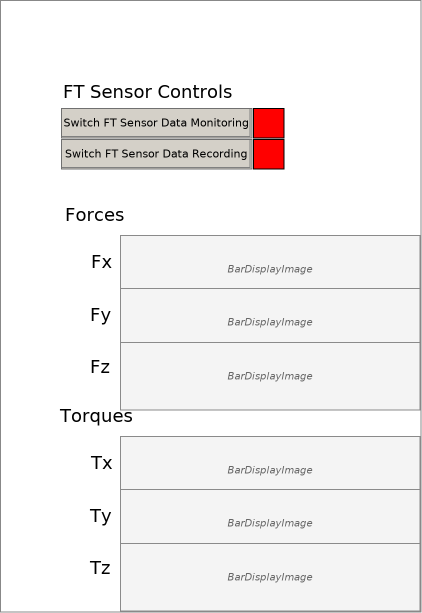
VISUALIZATION ForceAndTorque  // 422x613
    BarDisplayImage (120,235 300x68), value: Global.stFTData.Fx/10000, style: BarDisplayImage-Gray, scale format: %.1f, scale -5..5
        p518627256: Newtons (N)
    BarDisplayImage (120,288 300x68), value: Global.stFTData.Fy/10000, style: BarDisplayImage-Gray, scale format: %.1f, scale -5..5
        p518627256: Newtons (N)
    BarDisplayImage (120,342 300x68), value: Global.stFTData.Fz/10000, style: BarDisplayImage-Gray, scale format: %.1f, scale -5..5
        p518627256: Newtons (N)
    Label (88,247 34x30), "Fx"
    Label (87,300 34x30), "Fy"
    Label (87,352 34x30), "Fz"
    BarDisplayImage (120,436 300x68), value: Global.stFTData.Tx/100000, style: BarDisplayImage-Gray, scale format: %.1f, scale -1..1
        p518627256: Newton-meter (N-m)
    BarDisplayImage (120,489 300x68), value: Global.stFTData.Ty/100000, style: BarDisplayImage-Gray, scale format: %.1f, scale -1..1
        p518627256: Newton-meter (N-m)
    BarDisplayImage (120,543 300x68), value: Global.stFTData.Tz/100000, style: BarDisplayImage-Gray, scale format: %.1f, scale -1..1
        p518627256: Newton-meter (N-m)
    Label (88,448 34x30), "Tx"
    Label (87,501 34x30), "Ty"
    Label (87,553 34x30), "Tz"
    Label (62,197 98x36), "Forces"
    Label (57,398 98x36), "Torques"
    Button (61,108 191x30), "Switch FT Sensor Data Monitoring"
        OnMouseClick: toggle Global.bActivateFTDataCollection
    Button (61,139 191x30), "Switch FT Sensor Data Recording"
        OnMouseClick: toggle Global.bActivateFTDataRecording
    Rectangle (253,108 31x30), colour toggle: Global.bActivateFTDataCollection
    Rectangle (253,139 31x30), colour toggle: Global.bActivateFTDataRecording
    Label (60,77 246x30), "FT Sensor Controls"
END_VISUALIZATION

(* stored: Version 1.1.0.1, ProductVersion 3.1.4020.12
   Visu ForceAndTorque: Id {05bcde3d-23d3-4ede-9607-be1f3b0a538d} *)
